(*
Allows registration of FB implementing `I_Init`. 
*)
FUNCTION_BLOCK FINAL Init IMPLEMENTS I_InitNode, I_Debug
VAR
	_iInit			: I_Init;
	_iNext			: I_InitNode;
	_nState			: Result;
	_nPhase			: INT;
END_VAR

METHOD INTERNAL Attach : Result
VAR_INPUT
	iInit			: I_InitNode;
END_VAR
VAR
	_iThis			: I_InitNode := THIS^;
END_VAR
IF iInit = 0 THEN
	NewDebug(THIS^, Param.INIT_INTERNAL_DEBUG_MODE, Tc2_Standard.CONCAT(__POUNAME(), ': Itf = 0!'));
	RETURN;
END_IF

IF _iThis <> _Runtime.iLastInit THEN
	NewDebug(THIS^, Param.INIT_INTERNAL_DEBUG_MODE, Tc2_Standard.CONCAT(__POUNAME(), ': Is not the last node!'));
	RETURN;
END_IF

IF IsSome(iInit.state) THEN
	NewDebug(iInit, Param.INIT_INTERNAL_DEBUG_MODE, Tc2_Standard.CONCAT(__POUNAME(), ': Has already been added!'));
	RETURN;
END_IF

_Runtime.iLastInit := iInit;
_iNext := iInit;
END_METHOD

//FB_Init is always available implicitly and it is used primarily for initialization.
//The return value is not evaluated. For a specific influence, you can also declare the
//methods explicitly and provide additional code there with the standard initialization
//code. You can evaluate the return value.
{attribute 'hide'}
METHOD FB_Init: BOOL
VAR_INPUT
    bInitRetains: BOOL; // TRUE: the retain variables are initialized (reset warm / reset cold)
    bInCopyCode: BOOL;  // TRUE: the instance will be copied to the copy code afterward (online change)
	
	iInit			: I_Init;
END_VAR
IF IsSome(_nState) THEN
	RETURN;
END_IF

IF (_iInit := iInit) = 0 THEN
	_nState := Err.Itf0;
	NewDebug(THIS^, Param.INIT_INTERNAL_DEBUG_MODE, Tc2_Standard.CONCAT(__POUNAME(), ': Itf = 0!'));
	RETURN;
END_IF



IF _Runtime.iLastInit <> 0 THEN
	IF IsErr(_Runtime.iLastInit.Attach(THIS^), nOut => _nState) THEN
		NewDebug(THIS^, Param.INIT_INTERNAL_DEBUG_MODE, Tc2_Standard.CONCAT(__POUNAME(), ': Error inside!'));
	END_IF
ELSE
	_Runtime.iFirstInit := THIS^;
	_Runtime.iLastInit := THIS^;
	_nState := Ok;
END_IF
END_METHOD

METHOD INTERNAL Init
VAR_OUTPUT
	iNext: I_InitNode;
END_VAR
_iInit.Init(_nPhase);
iNext := _iNext;
END_METHOD

PROPERTY Phase : INT
GET
Phase := _nPhase;
END_GET
SET
_nPhase := Phase;
END_SET
END_PROPERTY

PROPERTY INTERNAL State : Result
GET
State := _nState;
END_GET
SET
IF IsNone(_nState) THEN
	_nState := State;
END_IF
END_SET
END_PROPERTY

END_FUNCTION_BLOCK

(* stored: Version 1.1.0.1
   POU Init: Id {f6ff46b8-b91f-4756-bbc4-c1b623301543}, SpecialFunc None
   Method Attach: Id {b570c3f9-4ba5-47de-92e9-c44911fd4d0b}
   Method FB_init: Id {a2ebe92c-4282-41f0-8dea-bb65a3d430c8}
   Method Init: Id {8876f358-5cbf-4b42-b262-c64dff58b017}
   Property Phase: Id {f49efe92-0704-4b7a-bf33-033e2ee1f8b6}
   Get Get: Id {c76d8319-3f16-4daf-83f6-feea49ac2dfa}
   Set Set: Id {bf1fdecc-4692-486c-ba82-57f3071cbc70}
   Property State: Id {f5ac33ac-0981-47a4-a9cd-9582eec70141}
   Get Get: Id {c6141bbd-407e-45af-a2fc-16001bb9949e}
   Set Set: Id {04dbdaec-18c9-4eca-95ab-24d03a281356} *)
